// Mitsubishi GX Works2 project: Ex02   PLC: Q02/Q02H

PROGRAM MAIN
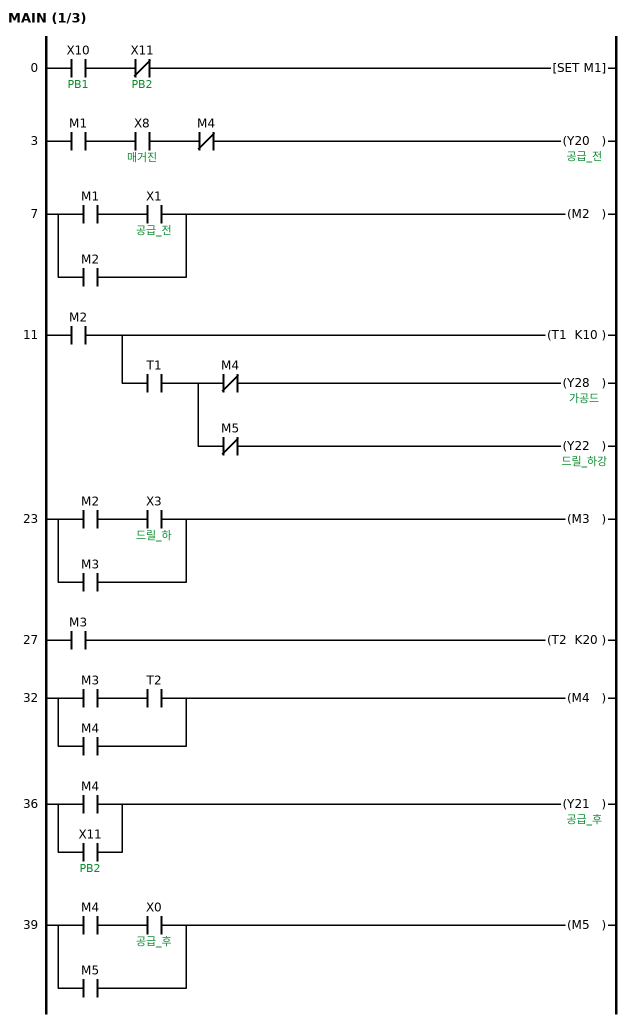
0     LD      X10  ; PB1
      ANI     X11  ; PB2
      SET     M1
3     LD      M1
      AND     X8  ; 매거진
      ANI     M4
      OUT     Y20  ; 공급_전
7     LD      M1
      AND     X1  ; 공급_전
      OR      M2
      OUT     M2
11    LD      M2
      OUT     T1 K10
      AND     T1
      MPS
      ANI     M4
      OUT     Y28  ; 가공드
      MPP
      ANI     M5
      OUT     Y22  ; 드릴_하강
23    LD      M2
      AND     X3  ; 드릴_하
      OR      M3
      OUT     M3
27    LD      M3
      OUT     T2 K20
32    LD      M3
      AND     T2
      OR      M4
      OUT     M4
36    LD      M4
      OR      X11  ; PB2
      OUT     Y21  ; 공급_후
39    LD      M4
      AND     X0  ; 공급_후
      OR      M5
      OUT     M5
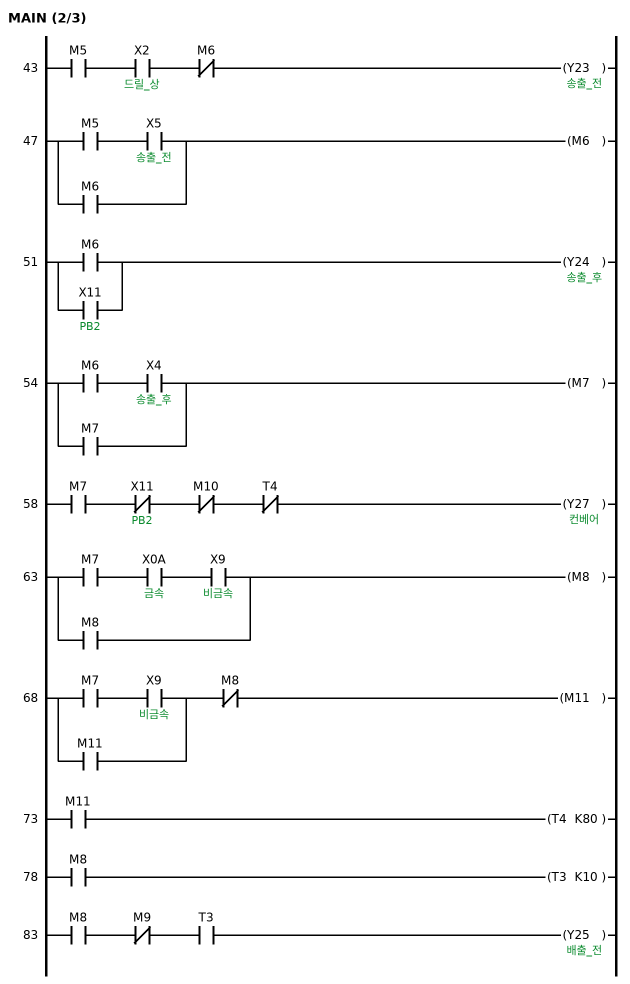
43    LD      M5
      AND     X2  ; 드릴_상
      ANI     M6
      OUT     Y23  ; 송출_전
47    LD      M5
      AND     X5  ; 송출_전
      OR      M6
      OUT     M6
51    LD      M6
      OR      X11  ; PB2
      OUT     Y24  ; 송출_후
54    LD      M6
      AND     X4  ; 송출_후
      OR      M7
      OUT     M7
58    LD      M7
      ANI     X11  ; PB2
      ANI     M10
      ANI     T4
      OUT     Y27  ; 컨베어
63    LD      M7
      AND     X0A  ; 금속
      AND     X9  ; 비금속
      OR      M8
      OUT     M8
68    LD      M7
      AND     X9  ; 비금속
      OR      M11
      ANI     M8
      OUT     M11
73    LD      M11
      OUT     T4 K80
78    LD      M8
      OUT     T3 K10
83    LD      M8
      ANI     M9
      AND     T3
      OUT     Y25  ; 배출_전
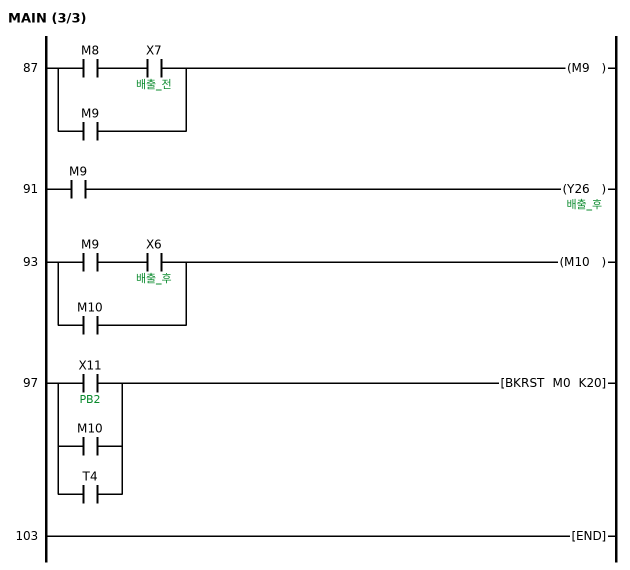
87    LD      M8
      AND     X7  ; 배출_전
      OR      M9
      OUT     M9
91    LD      M9
      OUT     Y26  ; 배출_후
93    LD      M9
      AND     X6  ; 배출_후
      OR      M10
      OUT     M10
97    LD      X11  ; PB2
      OR      M10
      OR      T4
      BKRST   M0 K20
103   END
END_PROGRAM

// device comments not shown above
X12  ; PB3
Y29  ; 적색
Y2A  ; 황색
Y2B  ; 녹색
